PROGRAM MAIN
VAR
	Axis_1 			: AXIS_REF;
	fbPower 		: MC_Power;
	bPower	 		: BOOL;
	
	fbMoveAbs 		: MC_MoveAbsolute;
	bMoveAbs 		: BOOL;	
	nPos 			: INT:=500;
	
	fbMoveRel 		: MC_MoveRelative;
	bMoveRel 		: BOOL;
	
	
	fbStop 			: MC_Stop; //acil durumlar için.
	bStop 			: BOOL; //bir kere true oldu mu false yapmadan eksen hareket etmez
	
	
	fbHalt 			: MC_Halt;//bir kere true oldu mu move fonksiyonlarından herhangi birine tekrar rising edge verirsek eksen hareket eder.
	bHalt 			: BOOL;
	
END_VAR

fbPower(
	Axis:= Axis_1, 
	Enable:=bPower , 
	Enable_Positive:=bPower , 
	Enable_Negative:=bPower , 
	Override:= 100, 
 );
 
 fbMoveAbs(
	Axis:=Axis_1 , 
	Execute:= bMoveAbs, 
	Position:= nPos, 
	Velocity:=100 , 
 );
 
 fbMoveRel(
	Axis:=Axis_1 , 
	Execute:=bMoveRel , 
	Distance:= 1000, 
	Velocity:= 500, 
 );

 fbStop(
	Axis:= Axis_1,
	Execute:=bStop);
	
fbHalt(
	Axis:=Axis_1 , 
	Execute:=bHalt , 
 );

END_PROGRAM

(* stored: Version 1.1.0.1, ProductVersion 3.1.4024.12
   POU MAIN: Id {a17149fd-3241-4a85-836c-fb039aca864f}, SpecialFunc None *)
